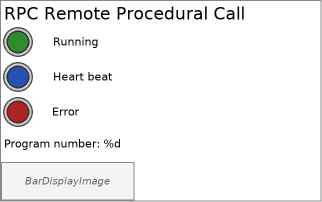
VISUALIZATION _VisuRPCStatusShow  // 322x202
    Lamp1 (1,25 34x34), variable: ComGVL._fbTryOutGetStatusRunning, style: Lamp-Lamp1-Green
    Rectangle (50,25 100x34), "Running"
    Label (1,1 319x25), "RPC Remote Procedural Call"
    Lamp1 (1,60 34x34), variable: ComGVL._fbTryOutGetStatusError, style: Lamp-Lamp1-Blue
    Rectangle (50,60 100x34), "Heart beat"
    Lamp1 (1,95 34x34), variable: ComGVL._fbTryOutGetStatusError, style: Lamp-Lamp1-Red
    Rectangle (49,95 100x34), "Error"
    BarDisplayImage (1,162 133x38), value: ComGVL._fbTryOutGetStatusProgress, style: BarDisplayImage-Gray, scale format: %.1f, scale 0..100
    Rectangle (1,130 176x28), "Program number: %d", text variable: ComGVL._fbTryOutGetStatusProgramNumber
END_VISUALIZATION

(* stored: Version 1.1.0.1, ProductVersion 3.1.4024.2
   Visu _VisuRPCStatusShow: Id {4f8b2118-2199-4c11-b93e-ce8a07b1717b} *)
